Omron CX-Programmer project NewProject (CX-Programmer 9.75)

# PLC NewPLC1: CP2E-N N

## Global symbols (name address type ; comment)
0.00 BOOL  ; Proxy Mie Kering 1
0.01 BOOL  ; STOP
0.02 BOOL  ; START BUTTON
0.03 BOOL  ; Proxy Mie Kering 2
0.04 BOOL  ; Proxy Mie Kering 3
0.05 BOOL  ; Proxy Mie Kering 4
0.06 BOOL  ; Proxy Mie Kering 5
0.07 BOOL  ; ProxyBowl1_FromMC
0.08 BOOL  ; ProxyBowl2_FromMC
0.09 BOOL  ; ProxyBowl3_FromMC
100.00 BOOL  ; Sole Mie 1
100.01 BOOL  ; Sole Mie 2
100.02 BOOL  ; Sole Mie 3
100.03 BOOL  ; Sole Mie 4
100.04 BOOL  ; Sole Mie 5
100.05 BOOL  ; Motor Cup Disp 1
100.06 BOOL  ; Motor Cup Disp 2
100.07 BOOL  ; Motor Cup Disp 3
101.00 BOOL  ; Sole Garnish
C005 BOOL  ; StockValidationCup
C006 BOOL  ; DispensedCup_cnt
C007 BOOL  ; Dispensed Mie Kering
C008 BOOL  ; StockValidationMie
D130 CHANNEL  ; Boiling Time Mie 1
D131 CHANNEL  ; Time to Pick Mie Kering 2
D132 CHANNEL  ; Time to pick Mie kering 3
D133 CHANNEL  ; Boiling Time Mie 2
D134 CHANNEL  ; Boiling Time Mie 3
D135 CHANNEL  ; Dispensing Timer
D140 CHANNEL  ; Time to Trigger Noodle 2 Disp
D141 CHANNEL  ; Time to Trigger Noodle 3 Disp
D30 CHANNEL  ; CupSelection
D31 CHANNEL  ; DispensedNoodle
D32 CHANNEL  ; NoodleSelector
D33 CHANNEL  ; Sisa Stock Mie
D34 CHANNEL  ; MinimumNoodle
D35 CHANNEL  ; Stock Cup
D36 CHANNEL  ; Sisa Cup Minimum
D5 CHANNEL  ; OrderQty (Local)
D6 CHANNEL  ; Order1_Menu (Local)
D7 CHANNEL  ; Order2_Menu (Local)
D8 CHANNEL  ; Order3_Menu (Local)
T000 BOOL  ; TIMER ActuatorMie
T001 BOOL  ; Cycle1 finish
T002 BOOL  ; Reset Second Cup
T003 BOOL  ; Rst Third Cup State
T004 BOOL  ; On MODBUS
T005 BOOL  ; TimerActuatorMie
T006 BOOL  ; Timer Boil Mie 1
T007 BOOL  ; Timer Pick Mie Kering 2
T008 BOOL  ; Timer Pick Mie Kering 3
T009 BOOL  ; Timer Boil Mie 2
T010 BOOL  ; Timer Boil Mie 3
T011 BOOL  ; Timer Actuator Mie 1
T012 BOOL  ; Timer Actuator Mie 2
T013 BOOL  ; Timer Actuator Mie 3
T014 BOOL  ; Timer Actuator Mie 4
T015 BOOL  ; Timer Actuator Mie 5
T016 BOOL  ; Timer CupDisp1
T017 BOOL  ; Timer CupDisp 3
T018 BOOL  ; Timer CupDisp3
T020 BOOL  ; Triger Noodle Disp
T021 BOOL  ; Trigger Noodle Disp
W100.01 BOOL  ; Finished Order From Robot
W100.02 BOOL  ; Garnish_on
W100.03 BOOL  ; Boiling_Mie1
W100.04 BOOL  ; Boiling_Mie2
W100.05 BOOL  ; Boiling_Mie3
W100.06 BOOL  ; RebusMie1_Done
W100.07 BOOL  ; RebusMie2_Done
W100.08 BOOL  ; RebusMie3_Done
W100.09 BOOL  ; Start Pick Mie 2 Kering
W100.10 BOOL  ; Start Pick Mie 3 Kering
W101.00 BOOL  ; MieKering1_Ready
W101.01 BOOL  ; MieKering2_Ready
W101.02 BOOL  ; MieKering3_Ready
W101.03 BOOL  ; MieKering4_Ready
W101.04 BOOL  ; MieKering5_Ready
W101.05 BOOL  ; Cup1 Ready
W101.06 BOOL  ; Cup2 Ready
W101.07 BOOL  ; Cup3 Ready
W101.08 BOOL  ; STOCK CUP HABIS
W102.08 BOOL  ; STOCK MIE HABIS
W103.00 BOOL  ; Dispensing ERROR
W103.01 BOOL  ; Reset Stock
W21.00 BOOL  ; ModbusOnCoil
W22.01 BOOL  ; Inc_Cup
W22.02 BOOL  ; Inc_Mie
W30.00 BOOL  ; ProxyBowl1_Inverted
W30.01 BOOL  ; ProxyBowl2_Inverted
W30.02 BOOL  ; ProxyBowl3_Inverted
W30.03 BOOL  ; Cup3_State
W31.00 BOOL  ; Inv_ProxyMie1
W31.01 BOOL  ; Inv_ProxyMie2
W31.02 BOOL  ; Inv_ProxyMie3
W31.03 BOOL  ; Inv_ProxyMie4
W31.04 BOOL  ; Inv_ProxyMie5
W31.05 BOOL  ; Mie5_State
W31.06 BOOL  ; ResetMie5
W31.07 BOOL  ; ResetCup3
W31.08 BOOL  ; LastMie
W32.00 BOOL  ; Sensor Mie Kosong
W32.01 BOOL  ; Sensor Cup Kosong
W32.02 BOOL  ; Garnish_State
W32.05 BOOL  ; Noodle Dispensed
W3.00 BOOL  ; StartRelay
W3.04 BOOL  ; Set Sensor
FB_MODBUSTCP_SERVER _CP2E003_ExecuteModTcpServer
Order1_Menu D110 CHANNEL  ; From PC
Order1_Topping1 D100 CHANNEL  ; From PC
Order1_Topping2 D101 CHANNEL  ; From PC
Order1_Topping3 D102 CHANNEL  ; From PC
Order2_Menu D111 CHANNEL  ; From PC
Order2_Topping1 D103 CHANNEL  ; From PC
Order2_Topping2 D104 CHANNEL  ; From PC
Order2_Topping3 D105 CHANNEL  ; From PC
Order3_Menu D112 CHANNEL  ; From PC
Order3_Topping1 D106 CHANNEL  ; From PC
Order3_Topping2 D107 CHANNEL  ; From PC
Order3_Topping3 D108 CHANNEL  ; From PC
Order_Quantity D120 CHANNEL  ; Order_Qty From PC
Start_Order W100.00 BOOL

## Program CookingMie (cyclic task 0)
Local symbols
p_LT BOOL
p_eq BOOL
p_gt BOOL
p_lt BOOL

### Section MODBUS

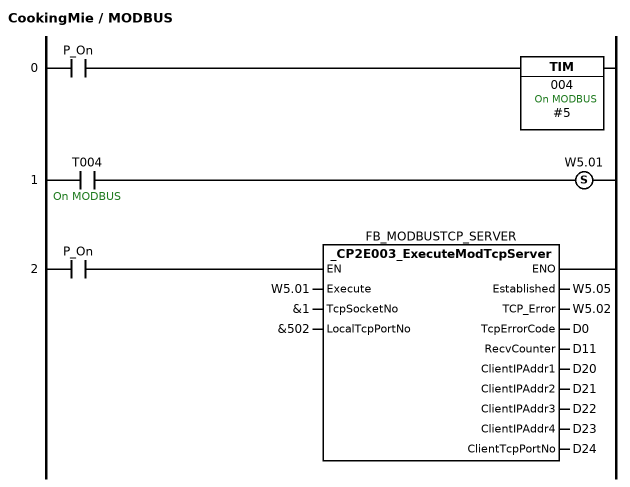
; rung 0
LD P_On
TIM 004 #5  ; On MODBUS
; rung 1
LD T004  ; On MODBUS
SET W5.01
; rung 2
LD P_On
CALL FB_MODBUSTCP_SERVER : _CP2E003_ExecuteModTcpServer (Execute := W5.01, TcpSocketNo := &1, LocalTcpPortNo := &502, Established => W5.05, TCP_Error => W5.02, TcpErrorCode => D0, RecvCounter => D11, ClientIPAddr1 => D20, ClientIPAddr2 => D21, ClientIPAddr3 => D22, ClientIPAddr4 => D23, ClientTcpPortNo => D24)

### Section Main

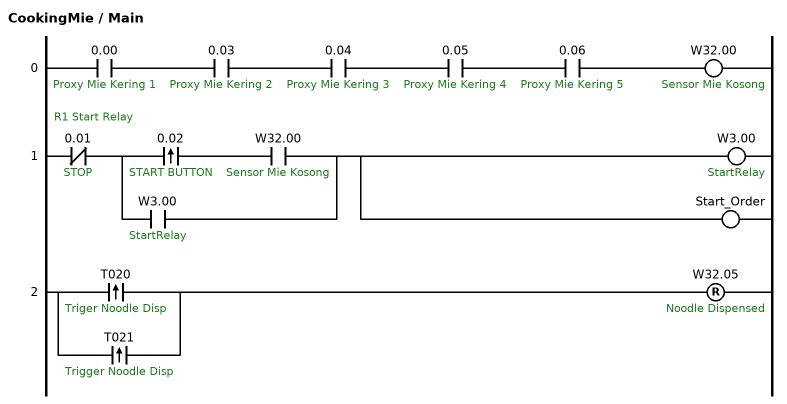
; rung 0
LD 0.00  ; Proxy Mie Kering 1
AND 0.03  ; Proxy Mie Kering 2
AND 0.04  ; Proxy Mie Kering 3
AND 0.05  ; Proxy Mie Kering 4
AND 0.06  ; Proxy Mie Kering 5
OUT W32.00  ; Sensor Mie Kosong
; rung 1: R1 Start Relay
LDNOT 0.01  ; STOP
@LD 0.02  ; START BUTTON
AND W32.00  ; Sensor Mie Kosong
OR W3.00  ; StartRelay
ANDLD
OUT W3.00  ; StartRelay
OUT Start_Order
; rung 2
@LD T020  ; Triger Noodle Disp
@OR T021  ; Trigger Noodle Disp
RSET W32.05  ; Noodle Dispensed

### Section Dispenser_Mie

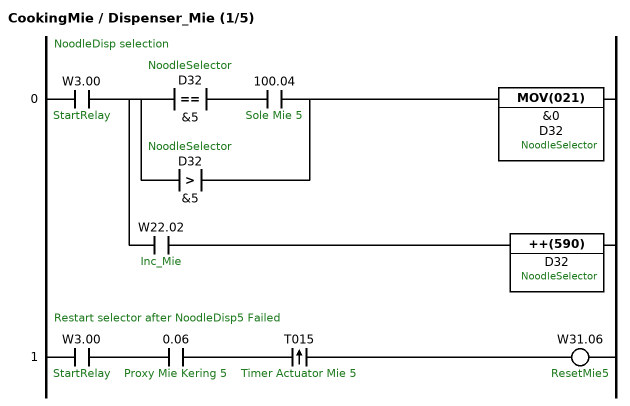
; rung 0: NoodleDisp selection
LD W3.00  ; StartRelay
OUT TR0
LD=(300) D32 &5  ; NoodleSelector
AND 100.04  ; Sole Mie 5
OR>(320) D32 &5  ; NoodleSelector
ANDLD
MOV(021) &0 D32  ; NoodleSelector
LD TR0
AND W22.02  ; Inc_Mie
++(590) D32  ; NoodleSelector
; rung 1: Restart selector after NoodleDisp5 Failed
LD W3.00  ; StartRelay
AND 0.06  ; Proxy Mie Kering 5
@AND T015  ; Timer Actuator Mie 5
OUT W31.06  ; ResetMie5

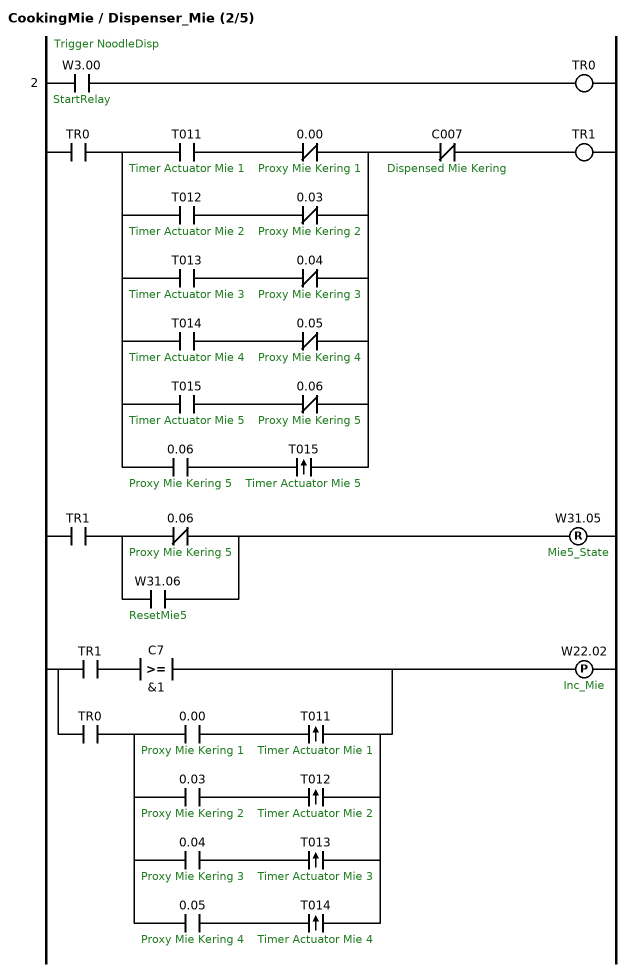
; rung 2: Trigger NoodleDisp
LD W3.00  ; StartRelay
OUT TR0
LD T011  ; Timer Actuator Mie 1
ANDNOT 0.00  ; Proxy Mie Kering 1
LD T012  ; Timer Actuator Mie 2
ANDNOT 0.03  ; Proxy Mie Kering 2
ORLD
LD T013  ; Timer Actuator Mie 3
ANDNOT 0.04  ; Proxy Mie Kering 3
ORLD
LD T014  ; Timer Actuator Mie 4
ANDNOT 0.05  ; Proxy Mie Kering 4
ORLD
LD T015  ; Timer Actuator Mie 5
ANDNOT 0.06  ; Proxy Mie Kering 5
ORLD
LD 0.06  ; Proxy Mie Kering 5
@AND T015  ; Timer Actuator Mie 5
ORLD
ANDLD
ANDNOT C007  ; Dispensed Mie Kering
OUT TR1
LDNOT 0.06  ; Proxy Mie Kering 5
OR W31.06  ; ResetMie5
ANDLD
RSET W31.05  ; Mie5_State
LD TR1
AND>=(325) C7 &1
LD TR0
LD 0.00  ; Proxy Mie Kering 1
@AND T011  ; Timer Actuator Mie 1
LD 0.03  ; Proxy Mie Kering 2
@AND T012  ; Timer Actuator Mie 2
ORLD
LD 0.04  ; Proxy Mie Kering 3
@AND T013  ; Timer Actuator Mie 3
ORLD
LD 0.05  ; Proxy Mie Kering 4
@AND T014  ; Timer Actuator Mie 4
ORLD
ANDLD
ORLD
DIFU(013) W22.02  ; Inc_Mie

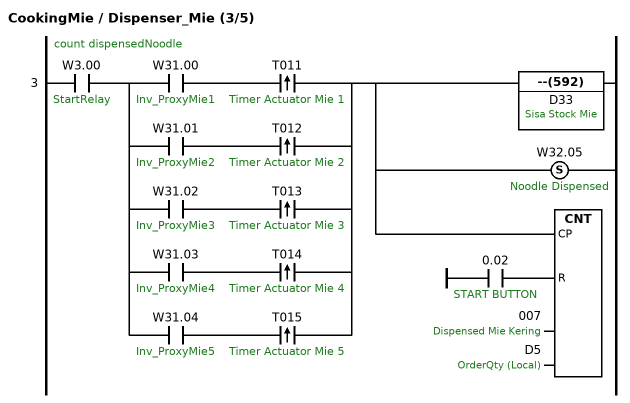
; rung 3: count dispensedNoodle
LD W3.00  ; StartRelay
LD W31.00  ; Inv_ProxyMie1
@AND T011  ; Timer Actuator Mie 1
LD W31.01  ; Inv_ProxyMie2
@AND T012  ; Timer Actuator Mie 2
ORLD
LD W31.02  ; Inv_ProxyMie3
@AND T013  ; Timer Actuator Mie 3
ORLD
LD W31.03  ; Inv_ProxyMie4
@AND T014  ; Timer Actuator Mie 4
ORLD
LD W31.04  ; Inv_ProxyMie5
@AND T015  ; Timer Actuator Mie 5
ORLD
ANDLD
--(592) D33  ; Sisa Stock Mie
SET W32.05  ; Noodle Dispensed
LD 0.02  ; START BUTTON
CNT 007 D5  ; OrderQty (Local), Dispensed Mie Kering

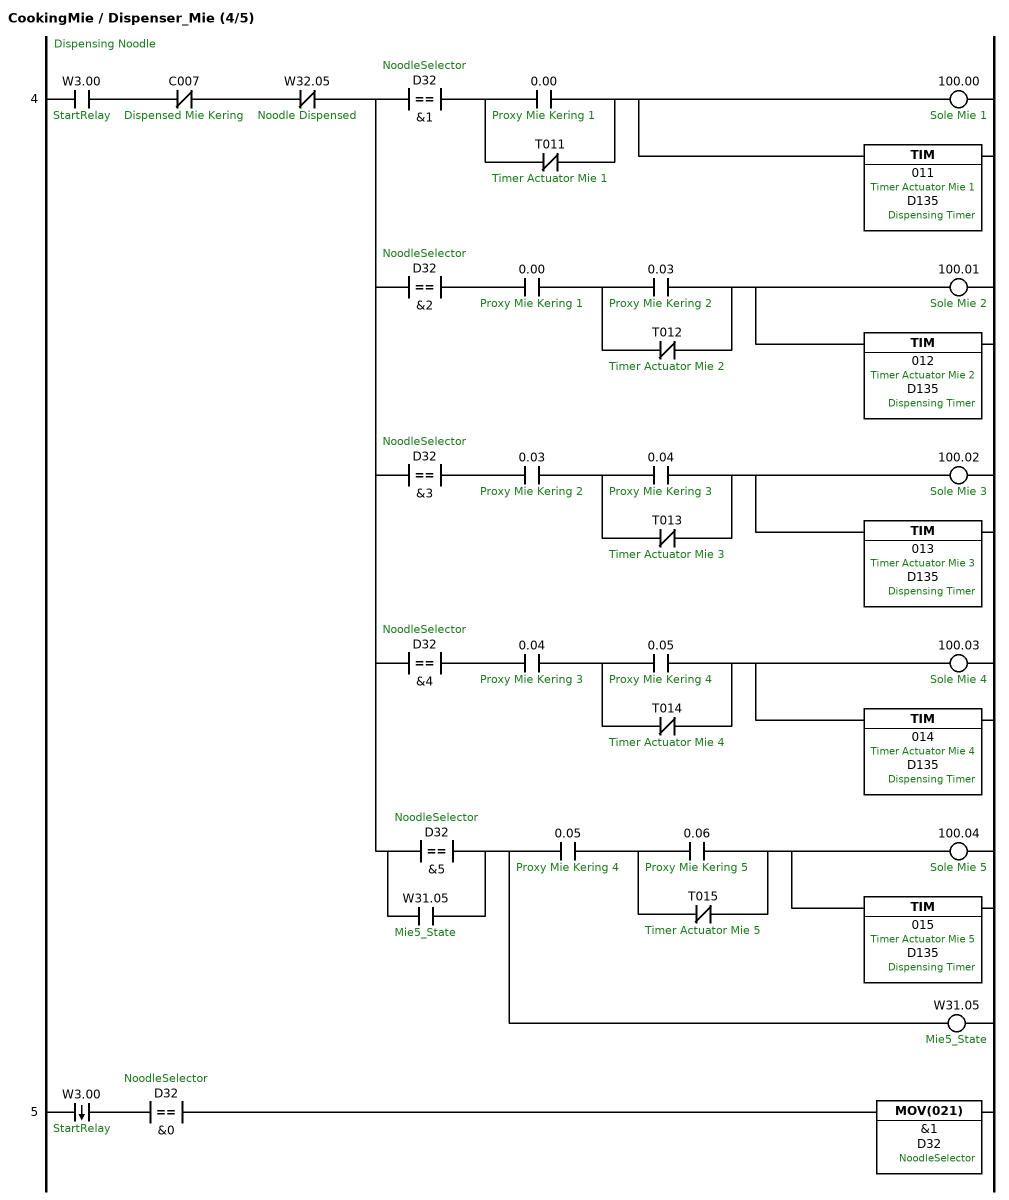
; rung 4: Dispensing Noodle
LD W3.00  ; StartRelay
ANDNOT C007  ; Dispensed Mie Kering
ANDNOT W32.05  ; Noodle Dispensed
OUT TR0
AND=(300) D32 &1  ; NoodleSelector
LD 0.00  ; Proxy Mie Kering 1
ORNOT T011  ; Timer Actuator Mie 1
ANDLD
OUT 100.00  ; Sole Mie 1
TIM 011 D135  ; Dispensing Timer, Timer Actuator Mie 1
LD TR0
AND=(300) D32 &2  ; NoodleSelector
AND 0.00  ; Proxy Mie Kering 1
LD 0.03  ; Proxy Mie Kering 2
ORNOT T012  ; Timer Actuator Mie 2
ANDLD
OUT 100.01  ; Sole Mie 2
TIM 012 D135  ; Dispensing Timer, Timer Actuator Mie 2
LD TR0
AND=(300) D32 &3  ; NoodleSelector
AND 0.03  ; Proxy Mie Kering 2
LD 0.04  ; Proxy Mie Kering 3
ORNOT T013  ; Timer Actuator Mie 3
ANDLD
OUT 100.02  ; Sole Mie 3
TIM 013 D135  ; Dispensing Timer, Timer Actuator Mie 3
LD TR0
AND=(300) D32 &4  ; NoodleSelector
AND 0.04  ; Proxy Mie Kering 3
LD 0.05  ; Proxy Mie Kering 4
ORNOT T014  ; Timer Actuator Mie 4
ANDLD
OUT 100.03  ; Sole Mie 4
TIM 014 D135  ; Dispensing Timer, Timer Actuator Mie 4
LD TR0
LD=(300) D32 &5  ; NoodleSelector
OR W31.05  ; Mie5_State
ANDLD
OUT TR0
AND 0.05  ; Proxy Mie Kering 4
LD 0.06  ; Proxy Mie Kering 5
ORNOT T015  ; Timer Actuator Mie 5
ANDLD
OUT 100.04  ; Sole Mie 5
TIM 015 D135  ; Dispensing Timer, Timer Actuator Mie 5
LD TR0
OUT W31.05  ; Mie5_State
; rung 5
%LD W3.00  ; StartRelay
AND=(300) D32 &0  ; NoodleSelector
MOV(021) &1 D32  ; NoodleSelector

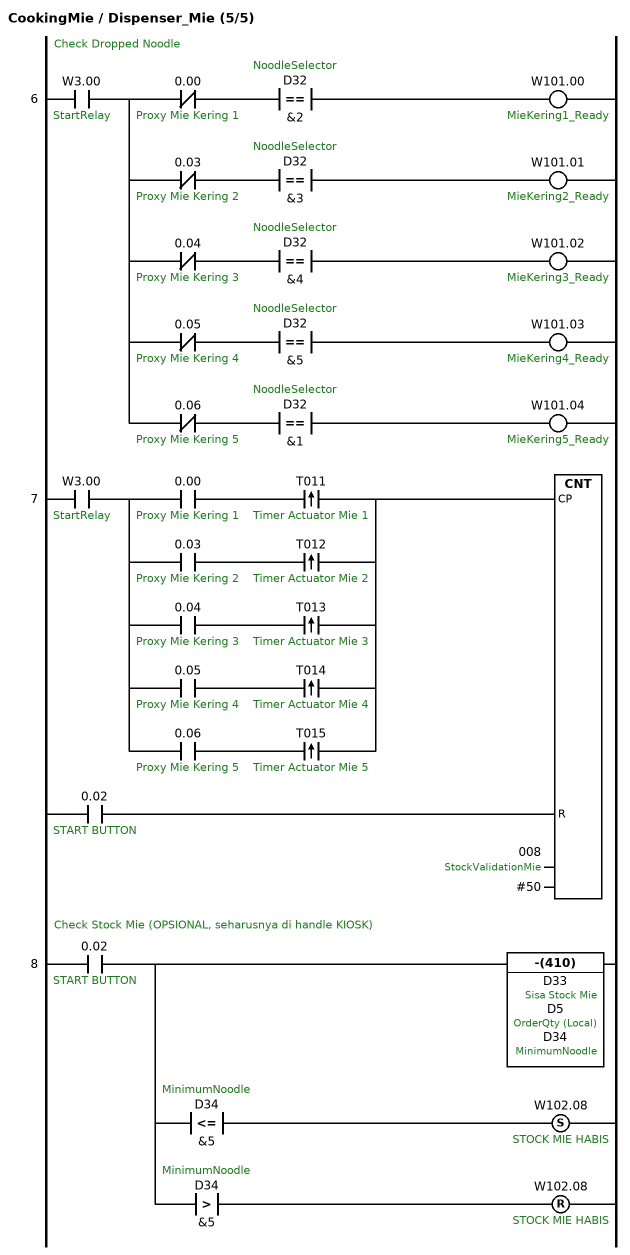
; rung 6: Check Dropped Noodle
LD W3.00  ; StartRelay
OUT TR0
ANDNOT 0.00  ; Proxy Mie Kering 1
AND=(300) D32 &2  ; NoodleSelector
OUT W101.00  ; MieKering1_Ready
LD TR0
ANDNOT 0.03  ; Proxy Mie Kering 2
AND=(300) D32 &3  ; NoodleSelector
OUT W101.01  ; MieKering2_Ready
LD TR0
ANDNOT 0.04  ; Proxy Mie Kering 3
AND=(300) D32 &4  ; NoodleSelector
OUT W101.02  ; MieKering3_Ready
LD TR0
ANDNOT 0.05  ; Proxy Mie Kering 4
AND=(300) D32 &5  ; NoodleSelector
OUT W101.03  ; MieKering4_Ready
LD TR0
ANDNOT 0.06  ; Proxy Mie Kering 5
AND=(300) D32 &1  ; NoodleSelector
OUT W101.04  ; MieKering5_Ready
; rung 7
LD W3.00  ; StartRelay
LD 0.00  ; Proxy Mie Kering 1
@AND T011  ; Timer Actuator Mie 1
LD 0.03  ; Proxy Mie Kering 2
@AND T012  ; Timer Actuator Mie 2
ORLD
LD 0.04  ; Proxy Mie Kering 3
@AND T013  ; Timer Actuator Mie 3
ORLD
LD 0.05  ; Proxy Mie Kering 4
@AND T014  ; Timer Actuator Mie 4
ORLD
LD 0.06  ; Proxy Mie Kering 5
@AND T015  ; Timer Actuator Mie 5
ORLD
ANDLD
LD 0.02  ; START BUTTON
CNT 008 #50  ; StockValidationMie
; rung 8: Check Stock Mie (OPSIONAL, seharusnya di handle KIOSK)
LD 0.02  ; START BUTTON
OUT TR0
-(410) D33 D5 D34  ; Sisa Stock Mie, OrderQty (Local), MinimumNoodle
AND<=(315) D34 &5  ; MinimumNoodle
SET W102.08  ; STOCK MIE HABIS
LD TR0
AND>(320) D34 &5  ; MinimumNoodle
RSET W102.08  ; STOCK MIE HABIS

### Section Dispenser_Cup

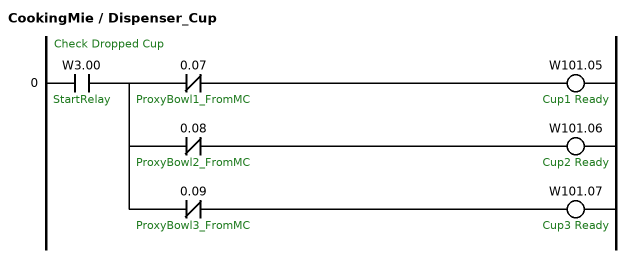
; rung 0: Check Dropped Cup
LD W3.00  ; StartRelay
OUT TR0
ANDNOT 0.07  ; ProxyBowl1_FromMC
OUT W101.05  ; Cup1 Ready
LD TR0
ANDNOT 0.08  ; ProxyBowl2_FromMC
OUT W101.06  ; Cup2 Ready
LD TR0
ANDNOT 0.09  ; ProxyBowl3_FromMC
OUT W101.07  ; Cup3 Ready

### Section Cooking_Process

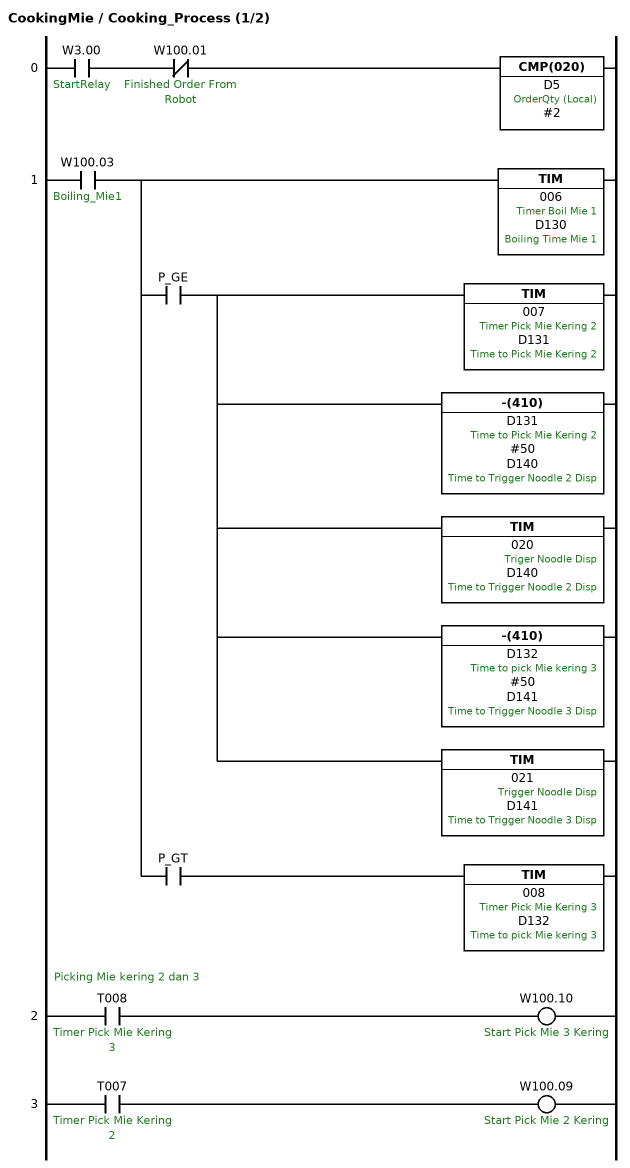
; rung 0
LD W3.00  ; StartRelay
ANDNOT W100.01  ; Finished Order From Robot
CMP(020) D5 #2  ; OrderQty (Local)
; rung 1
LD W100.03  ; Boiling_Mie1
OUT TR0
TIM 006 D130  ; Boiling Time Mie 1, Timer Boil Mie 1
AND P_GE
TIM 007 D131  ; Time to Pick Mie Kering 2, Timer Pick Mie Kering 2
-(410) D131 #50 D140  ; Time to Pick Mie Kering 2, Time to Trigger Noodle 2 Disp
TIM 020 D140  ; Time to Trigger Noodle 2 Disp, Triger Noodle Disp
-(410) D132 #50 D141  ; Time to pick Mie kering 3, Time to Trigger Noodle 3 Disp
TIM 021 D141  ; Time to Trigger Noodle 3 Disp, Trigger Noodle Disp
LD TR0
AND P_GT
TIM 008 D132  ; Time to pick Mie kering 3, Timer Pick Mie Kering 3
; rung 2: Picking Mie kering 2 dan 3
LD T008  ; Timer Pick Mie Kering 3
OUT W100.10  ; Start Pick Mie 3 Kering
; rung 3
LD T007  ; Timer Pick Mie Kering 2
OUT W100.09  ; Start Pick Mie 2 Kering

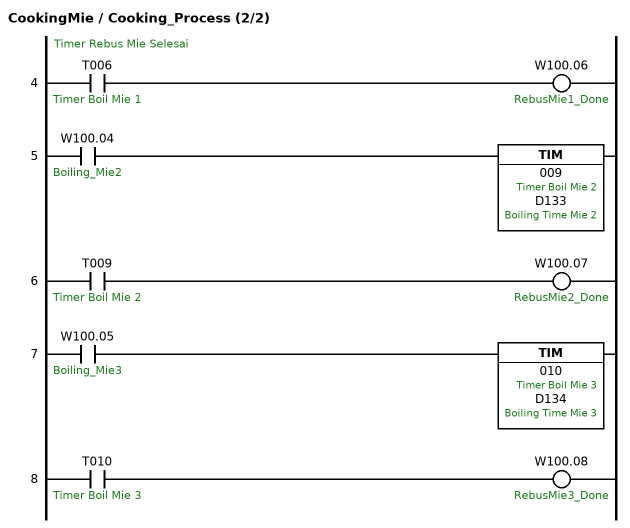
; rung 4: Timer Rebus Mie Selesai
LD T006  ; Timer Boil Mie 1
OUT W100.06  ; RebusMie1_Done
; rung 5
LD W100.04  ; Boiling_Mie2
TIM 009 D133  ; Boiling Time Mie 2, Timer Boil Mie 2
; rung 6
LD T009  ; Timer Boil Mie 2
OUT W100.07  ; RebusMie2_Done
; rung 7
LD W100.05  ; Boiling_Mie3
TIM 010 D134  ; Boiling Time Mie 3, Timer Boil Mie 3
; rung 8
LD T010  ; Timer Boil Mie 3
OUT W100.08  ; RebusMie3_Done

### Section Order_Settings

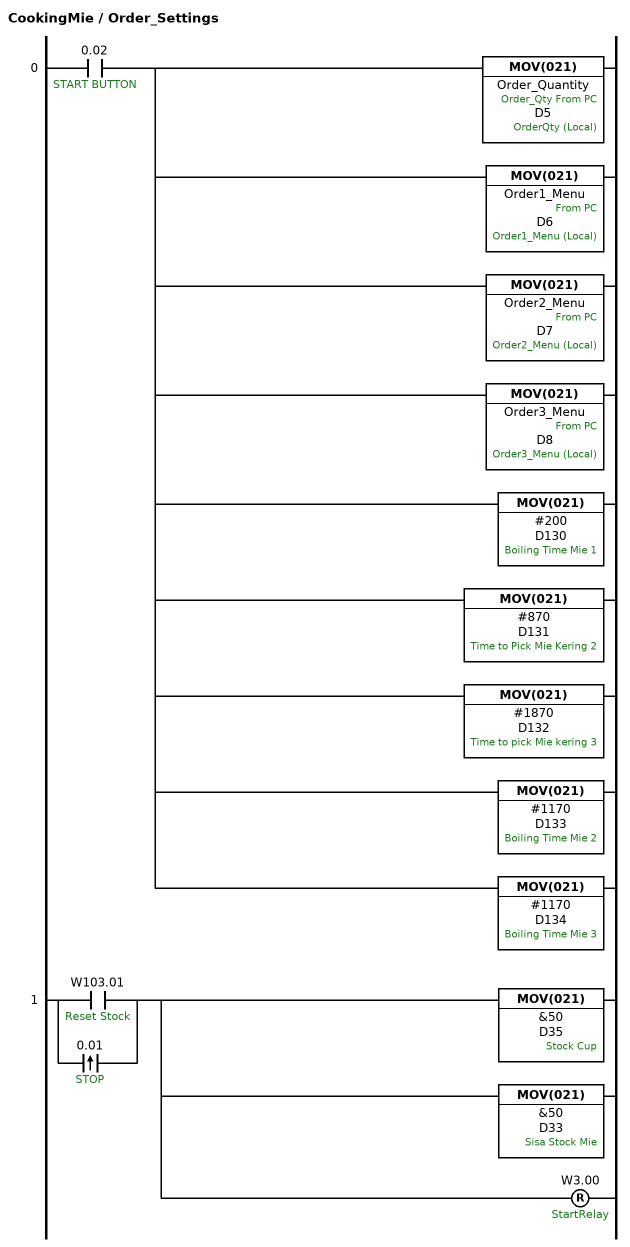
; rung 0
LD 0.02  ; START BUTTON
MOV(021) Order_Quantity D5  ; Order_Qty From PC, OrderQty (Local)
MOV(021) Order1_Menu D6  ; From PC, Order1_Menu (Local)
MOV(021) Order2_Menu D7  ; From PC, Order2_Menu (Local)
MOV(021) Order3_Menu D8  ; From PC, Order3_Menu (Local)
MOV(021) #200 D130  ; Boiling Time Mie 1
MOV(021) #870 D131  ; Time to Pick Mie Kering 2
MOV(021) #1870 D132  ; Time to pick Mie kering 3
MOV(021) #1170 D133  ; Boiling Time Mie 2
MOV(021) #1170 D134  ; Boiling Time Mie 3
; rung 1
LD W103.01  ; Reset Stock
@OR 0.01  ; STOP
MOV(021) &50 D35  ; Stock Cup
MOV(021) &50 D33  ; Sisa Stock Mie
RSET W3.00  ; StartRelay

### Section RESET_States

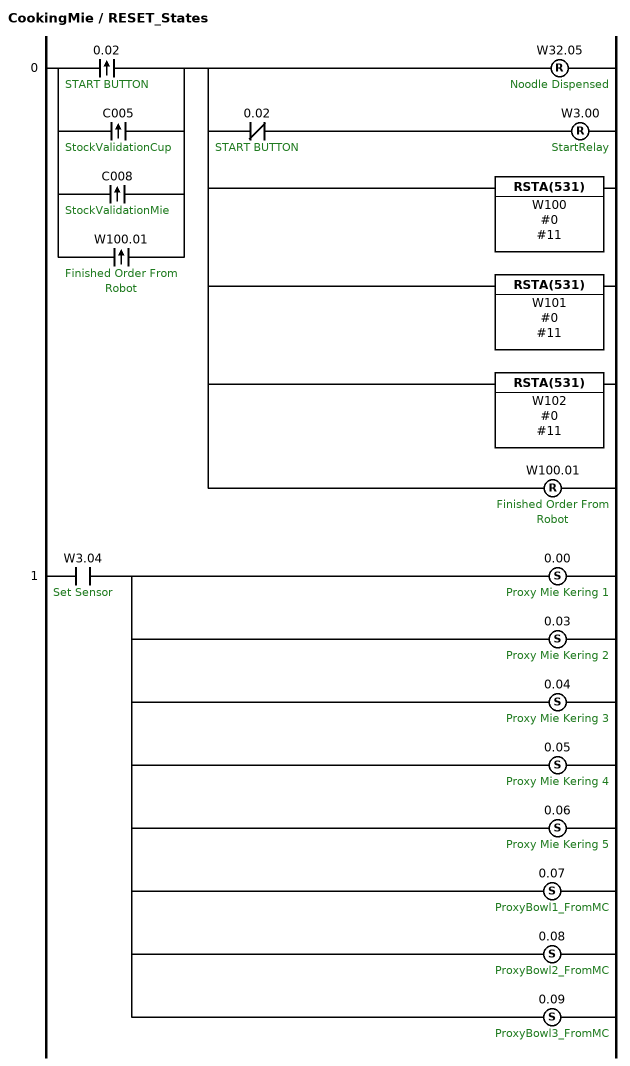
; rung 0
@LD 0.02  ; START BUTTON
@OR C005  ; StockValidationCup
@OR C008  ; StockValidationMie
@OR W100.01  ; Finished Order From Robot
OUT TR0
RSET W32.05  ; Noodle Dispensed
ANDNOT 0.02  ; START BUTTON
RSET W3.00  ; StartRelay
LD TR0
RSTA(531) W100 #0 #11
RSTA(531) W101 #0 #11
RSTA(531) W102 #0 #11
RSET W100.01  ; Finished Order From Robot
; rung 1
LD W3.04  ; Set Sensor
SET 0.00  ; Proxy Mie Kering 1
SET 0.03  ; Proxy Mie Kering 2
SET 0.04  ; Proxy Mie Kering 3
SET 0.05  ; Proxy Mie Kering 4
SET 0.06  ; Proxy Mie Kering 5
SET 0.07  ; ProxyBowl1_FromMC
SET 0.08  ; ProxyBowl2_FromMC
SET 0.09  ; ProxyBowl3_FromMC

### Section Invert_Sensor

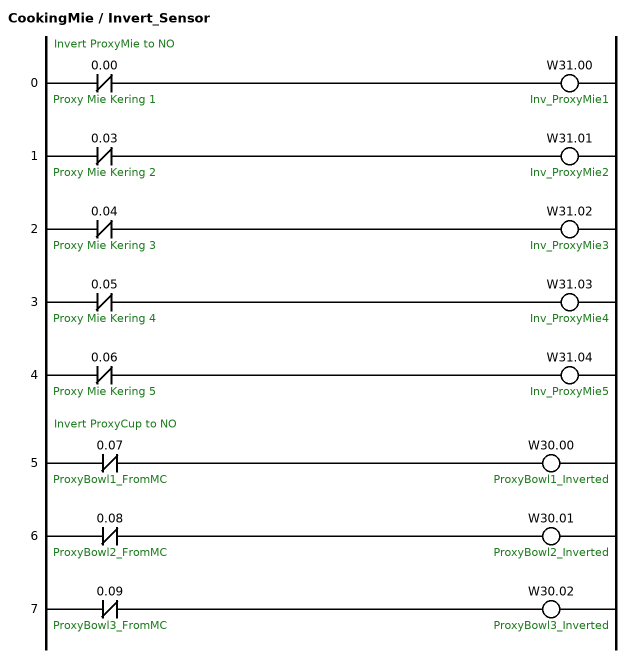
; rung 0: Invert ProxyMie to NO
LDNOT 0.00  ; Proxy Mie Kering 1
OUT W31.00  ; Inv_ProxyMie1
; rung 1
LDNOT 0.03  ; Proxy Mie Kering 2
OUT W31.01  ; Inv_ProxyMie2
; rung 2
LDNOT 0.04  ; Proxy Mie Kering 3
OUT W31.02  ; Inv_ProxyMie3
; rung 3
LDNOT 0.05  ; Proxy Mie Kering 4
OUT W31.03  ; Inv_ProxyMie4
; rung 4
LDNOT 0.06  ; Proxy Mie Kering 5
OUT W31.04  ; Inv_ProxyMie5
; rung 5: Invert ProxyCup to NO
LDNOT 0.07  ; ProxyBowl1_FromMC
OUT W30.00  ; ProxyBowl1_Inverted
; rung 6
LDNOT 0.08  ; ProxyBowl2_FromMC
OUT W30.01  ; ProxyBowl2_Inverted
; rung 7
LDNOT 0.09  ; ProxyBowl3_FromMC
OUT W30.02  ; ProxyBowl3_Inverted

### Section END
; rung 0
END(001)

## Function block _CP2E003_ExecuteModTcpServer (Omron library block, body left out)